SUBAPPLICATION Ventilsteuerung_Uebung_036 (* Spiegelabfolge V2 mit Schrittkette *)
  (* Standard: 61499-2 *)
  (* Version 1.0, 2023-10-23, franz *)
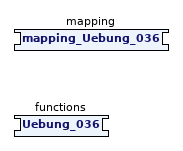
  SUBAPPS
    mapping : mapping_Uebung_036;
    functions : Uebung_036;
  END_SUBAPPS
END_SUBAPPLICATION
